(* signal debounce *)
FUNCTION_BLOCK FB_Debounce
VAR_INPUT
	bInput			: BOOL;		(* input signal from sensor that can show signal bounce *)
	tOnDelay		: TIME;		(* ON time of bInput before bOutput and bPulseOutput will be switched on *)
	tOffDelay		: TIME;		(* OFF time of bInput before bOutput will be switched off *)
	tPulseTime		: TIME;		(* ON time of bPulseOutput *)
END_VAR
VAR_OUTPUT
	bOutput			: BOOL;		(* output signal, follows bInput with ON and OFF delays to filter out signal bounce *)
	bPulseOutput	: BOOL;		(* pulse output signal, follows bInput with ON delay and stays on for specified pulse time *)
END_VAR
VAR
	fbOnDelay		: TON;
	fbOffDelay		: TON;
	fbDebounce		: SR;
	fbPulseTimer	: TP;
END_VAR
(*
-------------------------------------------------------------------------------------------------
Date		Version	Author	Comments
-------------------------------------------------------------------------------------------------
30/01/2015	3.00.00	PB		No change

-------------------------------------------------------------------------------------------------
02/07/2010	1.06.02	PB		Initial release

-------------------------------------------------------------------------------------------------
*)

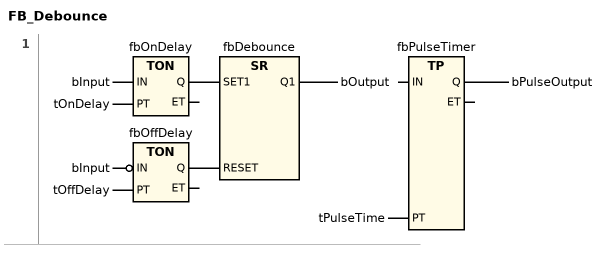
// NETWORK 1
fbOnDelay(IN := bInput, PT := tOnDelay); // TON
fbOffDelay(IN := NOT bInput, PT := tOffDelay); // TON
fbDebounce(SET1 := fbOnDelay.Q, RESET := fbOffDelay.Q); // SR
bOutput := fbDebounce.Q1;
fbPulseTimer(IN := fbDebounce.Q1, PT := tPulseTime); // TP
bPulseOutput := fbPulseTimer.Q;

END_FUNCTION_BLOCK

(* stored: Version 1.1.0.1, ProductVersion 3.1.4024.15
   POU FB_Debounce: Id {82a4d7df-c700-4d0e-9026-33be284f0812}, SpecialFunc None *)
